(* IEC 61131-3 sources: ATCMcontrol_Engineering/src/TargetBase/Libs/ATCM_Socket, 10 files *)

(* ---- SocketAccept.st ---- *)
(*[[
    UserURL= "ATCMfile:SocketAccept.htm"
]]*)
FUNCTION SocketAccept:DWORD

VAR_INPUT
   ListeningSocket: UDINT;
END_VAR

VAR_OUTPUT
   AcceptSocket:  UDINT;
END_VAR

inline {STDLIB(SocketAccept)}

END_FUNCTION

(* ---- SocketBind.st ---- *)
(*[[
    UserURL= "ATCMfile:SocketBind.htm"
]]*)
FUNCTION SocketBind:DWORD

VAR_INPUT
   Socket:        UDINT;
   SocketAddress: SocketAddressType;
END_VAR

inline {STDLIB(SocketBind)}

END_FUNCTION

(* ---- SocketClose.st ---- *)
(*[[
    UserURL= "ATCMfile:SocketClose.htm"
]]*)
FUNCTION SocketClose:DWORD

VAR_INPUT
   Socket:  UDINT;
END_VAR

inline {STDLIB(SocketClose)}

END_FUNCTION

(* ---- SocketConnect.st ---- *)
(*[[
    UserURL= "ATCMfile:SocketConnect.htm"
]]*)
FUNCTION SocketConnect:DWORD

VAR_INPUT
   Socket: UDINT;
   SocketAddress: SocketAddressType;
END_VAR

inline {STDLIB(SocketConnect)}

END_FUNCTION

(* ---- SocketCreate.st ---- *)
(*[[
    UserURL= "ATCMfile:SocketCreate.htm"
]]*)
FUNCTION SocketCreate:DWORD

VAR_INPUT
   AddressFamily:   DINT;
   ProtocolType:    DINT;
END_VAR

VAR_OUTPUT
   Socket:  UDINT;
END_VAR

inline {STDLIB(SocketCreate)}

END_FUNCTION

(* ---- SocketEnableNonblocking.st ---- *)
(*[[
    UserURL= "ATCMfile:SocketEnableNonblocking.htm"
]]*)
FUNCTION SocketEnableNonblocking:DWORD

VAR_INPUT
   Socket:  UDINT;
   NonblockingMode : BOOL;
END_VAR

inline {STDLIB(SocketEnableNonblocking)}

END_FUNCTION

(* ---- SocketListen.st ---- *)
(*[[
    UserURL= "ATCMfile:SocketListen.htm"
]]*)
FUNCTION SocketListen:DWORD

VAR_INPUT
   Socket:  UDINT;
   Backlog: DINT;
END_VAR

inline {STDLIB(SocketListen)}

END_FUNCTION

(* ---- SocketReceive.st ---- *)
(*[[
    UserURL= "ATCMfile:SocketReceive.htm"
]]*)
FUNCTION SocketReceive:DWORD

VAR_INPUT
   Socket:    UDINT;
END_VAR

VAR_OUTPUT
   Buffer:          ARRAY OF BYTE;
   ReceivedDataLen: DINT;
END_VAR

inline {STDLIB(SocketReceive)}

END_FUNCTION

(* ---- SocketSelect.st ---- *)
(*[[
    UserURL= "ATCMfile:SocketSelect.htm"
]]*)
FUNCTION SocketSelect:DWORD

VAR_INPUT
   Socket:    UDINT;
   Timeout:   INT;
END_VAR

VAR_OUTPUT
	Status:   UINT;
END_VAR

inline {STDLIB(SocketSelect)}

END_FUNCTION

(* ---- SocketSend.st ---- *)
(*[[
    UserURL= "ATCMfile:SocketSend.htm"
]]*)
FUNCTION SocketSend:DWORD

VAR_INPUT
   Socket:  UDINT;
   Data:    ARRAY OF BYTE;
   DataLen: DINT;
   DestinationAddress: SocketAddressType;
END_VAR

VAR_OUTPUT
   SentDataLen:  DINT;
END_VAR

inline {STDLIB(SocketSend)}

END_FUNCTION
